// TIA Portal V16 export
// export: Created 2021-09-08T12:46:15.8906042Z, ExportSetting WithDefaults, DisplayName Totally Integrated Automation Portal, DisplayVersion V16 Update 3, DisplayName TIA Portal Version Control Interface, DisplayVersion V16 Update 2, DisplayName TIA Portal Openness, DisplayVersion V16 Update 3, DisplayName TIA Portal Teamcenter Gateway, DisplayVersion V16, DisplayName STEP 7 Professional, DisplayVersion V16 Update 3, DisplayName STEP 7 Safety, DisplayVersion V16, DisplayName WinCC Advanced, DisplayVersion V16 Update 3
TYPE "setPID"
// stored: IsFailsafeCompliant false
   STRUCT
      spAuto { S7_SetPoint := 'True'} : Real;
      spHand : Real;
      TI { S7_SetPoint := 'True'} : Real := 10.0;
      Gain { S7_SetPoint := 'True'} : Real := 2.0;
      min { S7_SetPoint := 'True'} : Real := 30.0;
      max { S7_SetPoint := 'True'} : Real := 100.0;
      dead { S7_SetPoint := 'True'} : Real := 0.1;
      outPID : Real;
      cmFixSP : Bool;
      cmFreeze : Bool;
      cmStartSP : Bool;
      spareByte : Byte;
      fixSP { S7_SetPoint := 'True'} : Real;
      spStart : Real;
      spare_2 : DInt;
   END_STRUCT;
END_TYPE
